Fanuc KAREL source: ka00133.KL

-- PROVISIONAL review KL for V770-1; original PC SHA256 30ebff037a6a41b73d09fdda58c1e1cfc6cd1c1c8f43bec7cbd895efdc7580f3
-- Incomplete behavior may be omitted. Consult companion uncertainty JSON. Do not deploy.
PROGRAM KA00133
%NOLOCKGROUP
VAR
  DST : INTEGER
-- UNRESOLVED_DECL SRC type=002017
BEGIN
  -- UNRESOLVED_PC offsets 5-19; opcodes 2E,22,9D,33,B4
  -- UNRESOLVED_PC offsets 24-39; opcodes 22,9D,33,B3,23
  -- UNRESOLVED_PC offsets 44-48; opcodes 7F
END KA00133
